(* Schneider Machine Expert - Basic project first try FIFO LIFO, file version 2.7.0.0 *)
(* ProjectInformations: Name=New project *)

HARDWARE
  Cpu 0: TM221M16R/G
  EthernetConfiguration: NetworkName=M221, IpAllocationMode=FixedAddress, IpAddress=0.0.0.0, SubnetMask=0.0.0.0
  SerialLineConfiguration: Baud=Baud19200, Parity=ParityEven, DataBits=DataBits8, StopBits=StopBits1, PhysicalMedium=PhysicalMediumRs485, TransmissionMode=TransmissionModeModbusRtu, SlaveId=1, Addressing=SlaveAddressing
  MastTask: UsePeriodScanMode=false, PeriodScan=100
  FastTask: Period=255
  CpuBehavior: StartingMode=StartAsPreviousState, AutoSaveRamOnEeprom=true, WatchdogPeriod=250

SYMBOLS  (address, symbol, comment, settings)
  %M10      PET_FIFO_RESET
  %M11      PET_FIFO_STORE
  %M12      PET_FIFO_RETRIEVE
  %M13      PET_FIFO_FREE
  %M14      PET_FIFO_FREEE
  %MW10     CFG_FIFO_NEW_VALUE
  %MW11     IND_FIFO_GET_VALUE
  %R0       INST_FIFO

POU New POU
  (* SectionNumber=1 *)

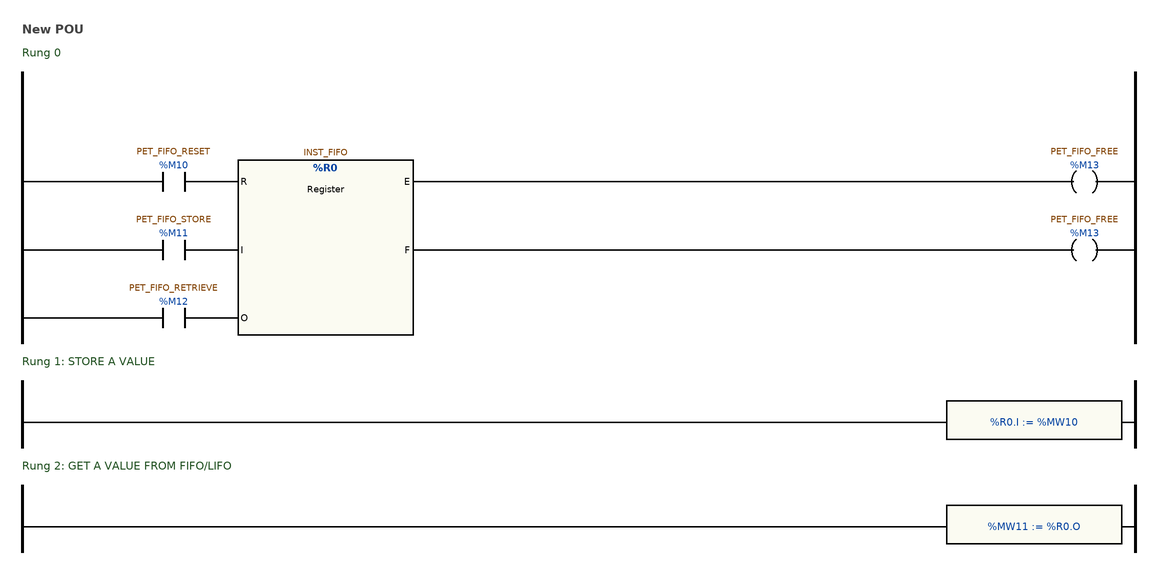

// Rung 0
  BLK %R0                 (* INST_FIFO *)
  LD %M10                 (* PET_FIFO_RESET *)
  R
  LD %M11                 (* PET_FIFO_STORE *)
  I
  LD %M12                 (* PET_FIFO_RETRIEVE *)
  O
  OUT_BLK
  LD E
  ST %M13                 (* PET_FIFO_FREE *)
  LD F
  ST %M13                 (* PET_FIFO_FREE *)
  END_BLK
  // as ST:
  //   INST_FIFO(R := PET_FIFO_RESET, I := PET_FIFO_STORE, O := PET_FIFO_RETRIEVE);
  //   PET_FIFO_FREE := INST_FIFO.E;
  //   PET_FIFO_FREE := INST_FIFO.F;

// Rung 1: STORE A VALUE
  LD 1
  [ %R0.I := %MW10 ]      (* INST_FIFO, CFG_FIFO_NEW_VALUE *)
  // as ST:
  //   INST_FIFO.I := CFG_FIFO_NEW_VALUE;

// Rung 2: GET A VALUE FROM FIFO/LIFO
  LD 1
  [ %MW11 := %R0.O ]      (* IND_FIFO_GET_VALUE, INST_FIFO *)
  // as ST:
  //   IND_FIFO_GET_VALUE := INST_FIFO.O;
